// TIA Portal project "Инвинтариаз_V1" (V16)

(* hardware
DEVICE "S7-1200 station_1"  S7-1200 Station
   slot 0: "Rack_0"  S7-1200 Rack  Rack  V1.0
   slot 1: "PLC_1"  CPU 1214C DC/DC/Rly  6ES7 214-1HG40-0XB0  V4.4
   slot 2: "AI 4xRTD_1"  SM 1231 AI4 x RTD  6ES7 231-5PD32-0XB0  V2.0
   slot 3: "AQ 4x14BIT_1"  6ES7 232-4HD32-0XB0  V2.1
*)

// ===== PLC "PLC_1"  CPU 1214C DC/DC/Rly =====

VAR_GLOBAL   // PLC tag table "Default tag table"
   "System_Byte" AT %MB1110 : Byte;
   "FirstScan" AT %M1110.0 : Bool;
   "DiagStatusUpdate" AT %M1110.1 : Bool;
   "AlwaysTRUE" AT %M1110.2 : Bool;
   "AlwaysFALSE" AT %M1110.3 : Bool;
   "Clock_Byte" AT %MB1000 : Byte;
   "Clock_10Hz" AT %M1000.0 : Bool;
   "Clock_5Hz" AT %M1000.1 : Bool;
   "Clock_2.5Hz" AT %M1000.2 : Bool;
   "Clock_2Hz" AT %M1000.3 : Bool;
   "Clock_1.25Hz" AT %M1000.4 : Bool;
   "Clock_1Hz" AT %M1000.5 : Bool;
   "Clock_0.625Hz" AT %M1000.6 : Bool;
   "Clock_0.5Hz" AT %M1000.7 : Bool;
END_VAR

VAR_GLOBAL   // PLC tag table "_Test"
   "Test_En" AT %M0.0 : Bool;
   "t_Lavel_1" AT %M0.1 : Bool;
   "t_Lavel_2" AT %M0.2 : Bool;
   "t_Wardrob1" AT %M0.3 : Bool;
   "t_Wardrob2" AT %M0.4 : Bool;
   "t_time" AT %MD2 : DInt;
   "t_Intemp1" AT %MD6 : Real;
   "t_Intemp_2" AT %MD10 : Real;
   "t_SetTemp" AT %MD14 : Real;
   "t_Set_Delta" AT %MD18 : Real;
   "t_startTime" AT %M0.5 : Bool;
   "t_SetTimer" AT %MD22 : DInt;
   "t_Point_Cold" AT %M0.6 : Bool;
   "t_Finish_Paster" AT %M0.7 : Bool;
   "t_Set_Temp_Cold" AT %MD26 : Real;
   "t_Speed_1" AT %MW30 : Int;
   "t_Speed_2" AT %MW32 : Int;
   "tPaster_St" AT %M1.0 : Bool;
   "tColder_Sr" AT %M1.1 : Bool;
   "t_start" AT %M1.2 : Bool;
   "t_Stop" AT %M1.3 : Bool;
   "t_Alarm" AT %M1.4 : Bool;
END_VAR

TYPE "Tipe_DI"
   STRUCT
      f_DI_out : Bool;
      "bFiltr_on/off" : Bool := true;   // Вкл/выкл фильтрацию входа
      diTime_filtr : Time := T#100ms;   // Уставка времени фильтрации
      bSimulation : Bool;   // Включение режима симуляции
      "bSim_On/Off" : Bool;   // Управление симуляцией
   END_STRUCT;
END_TYPE

DATA_BLOCK "FV_1"   // DB8
{ S7_Optimized_Access := 'FALSE' }
VERSION : 0.1
// stored: InstanceOfName Valve(c/o)
"Valve(c/o)"
BEGIN
END_DATA_BLOCK

DATA_BLOCK "fb_DI_St_DB_1"   // DB9
{ S7_Optimized_Access := 'TRUE' }
VERSION : 0.1
// stored: InstanceOfName fb_DI_St
"fb_DI_St"
BEGIN
END_DATA_BLOCK

DATA_BLOCK "fb_DI_St_DB"   // DB10
{ S7_Optimized_Access := 'TRUE' }
VERSION : 0.1
// stored: InstanceOfName fb_DI_St
"fb_DI_St"
BEGIN
END_DATA_BLOCK

DATA_BLOCK "fb_DI_St_DB_2"   // DB12
{ S7_Optimized_Access := 'TRUE' }
VERSION : 0.1
// stored: InstanceOfName fb_DI_St
"fb_DI_St"
BEGIN
END_DATA_BLOCK

// folder: DB_FB

DATA_BLOCK "Набор Воды_DB"   // DB1
{ S7_Optimized_Access := 'TRUE' }
VERSION : 0.1
// stored: InstanceOfName Набор Воды
"Набор Воды"
BEGIN
END_DATA_BLOCK

DATA_BLOCK "Гл_Блок_Шкафа_DB"   // DB2
{ S7_Optimized_Access := 'TRUE' }
VERSION : 0.1
// stored: InstanceOfName Гл_Блок_Шкафа
"Гл_Блок_Шкафа"
BEGIN
END_DATA_BLOCK

DATA_BLOCK "Контроль темп_DB"   // DB3
{ S7_Optimized_Access := 'TRUE' }
VERSION : 0.1
// stored: InstanceOfName Контроль темп
"Контроль темп"
BEGIN
END_DATA_BLOCK

DATA_BLOCK "Отсчет времени пастеризации_DB"   // DB4
{ S7_Optimized_Access := 'TRUE' }
VERSION : 0.1
// stored: InstanceOfName Отсчет времени пастеризации
"Отсчет времени пастеризации"
BEGIN
END_DATA_BLOCK

DATA_BLOCK "Охлаждение_DB"   // DB6
{ S7_Optimized_Access := 'TRUE' }
VERSION : 0.1
// stored: InstanceOfName Охлаждение
"Охлаждение"
BEGIN
END_DATA_BLOCK

DATA_BLOCK "Старт_DB"   // DB7
{ S7_Optimized_Access := 'TRUE' }
VERSION : 0.1
// stored: InstanceOfName Старт
"Старт"
BEGIN
END_DATA_BLOCK

// folder: HMI

DATA_BLOCK "DI_For_HMI"   // DB11
{ S7_Optimized_Access := 'FALSE' }
VERSION : 0.1
   VAR
      DI_0 : "Tipe_DI";
      DI_1 : "Tipe_DI";
      DI_2 : "Tipe_DI";
      DI_3 : "Tipe_DI";
      DI_4 : "Tipe_DI";
      DI_5 : "Tipe_DI";
      DI_6 : "Tipe_DI";
   END_VAR
BEGIN
END_DATA_BLOCK

// folder: R_trig

DATA_BLOCK "R_trig_Time1S"   // DB5
{ S7_Optimized_Access := 'TRUE' }
VERSION : 0.1
// stored: InstanceOfName R_trig
"R_trig"
BEGIN
END_DATA_BLOCK

// folder: (top level)

FUNCTION_BLOCK "Pump"   // FB1, SCL
{ S7_Optimized_Access := 'FALSE' }
VERSION : 0.1
   VAR_INPUT
      bManualMode : Bool;   // Выбор ручного режима
      bManualStart : Bool;   // Ручной режим - старт
      bManualStop : Bool;   // Ручной режим - стоп
      rManualSpeed : Real;   // Ручной режим - скорость
      bDryRunn : Bool;   // Защита от сухого хода
      bAutoSTop : Bool;   // Остановка насоса
      bAutoStartPerm : Bool;   // Команда на работоу в авто режиме
      rAutoSpeed : Real;   // Скорость в авто режиме
      bАвтоматы : Bool;   // Готовность привода (автоматы)
      bПускатели : Bool;   // Готовность Пускателя
      bDriveRunning : Bool;   // Привод в работе
      bDriveFault : Bool;   // Привод в ошибке
      rMinSpeed : Real;   // Минимальная скорость
      rMaxSpeed : Real := 100.0;   // Максимальная скорость
      bResetFault : Bool;   // Сброс аварии
   END_VAR
   VAR_OUTPUT
      bRunCmd : Bool;   // Пуск частотника
      iSpeedOut : Int;   // Скорость насоса для аналогового выхода
      "rSpeedHMI(0-100)" : Real;   // Скорость работы (0-100) для HMI
      bPumpRunning : Bool;   // Работа
      bPumpFault : Bool;   // Авария
      iStatus : Int;   // Статус (0 - стоп 1 - работа 2 - авария)
   END_VAR
   VAR
      bFaultLatch : Bool;
      bRunRequest : Bool;
      rSpeedPump : Real;   // Скорость насоса
      TON_NotStartRun : TON_TIME;   // ТАймер ожидания сигнала о запуске
      TON_NotContactRun : TON_TIME;   // ТАймер ожидания с контактора
      TON_DryRun : TON_TIME;   // Таймер сухого хода
   END_VAR
BEGIN
   (*
   // 1. Обработка аварий
   // Обработка ожидания сигнала о работе после старта
   IF #bAutoStartPerm THEN
       ;

   END_IF;
   *)

   // 1 Ручной режим
   IF #bManualMode THEN
       // Ручной режим
       IF #bManualStart AND NOT #bManualStop THEN
           #bRunRequest := TRUE;
       ELSIF #bManualStop THEN // OR NOT #bАвтоматы THEN
           #bRunRequest := FALSE;
       END_IF;
   ELSE
       // Автоматический режим
       // 
       //Обработка аварий
       //
       //Таймер ожидания останова по сухому ходу
       #TON_DryRun(IN := NOT #bDryRunn,
                   PT := t#1s);    //
       //--------------------------------------------------------------------------------------------------------
       IF #bAutoStartPerm AND NOT #bAutoSTop AND #bDryRunn THEN
           #TON_NotStartRun(IN := NOT #bDriveRunning AND #bDryRunn, PT := t#5s);  //Таймер ожидания сигнала подтверждения пуска от частотника
           #TON_NotContactRun(IN := NOT #bПускатели, PT := t#10s);  //Таймер ожидания сигнала подтверждения пуска от пускателя


       ELSE
           #TON_NotStartRun(IN :=FALSE,PT := t#5s);
           #TON_NotContactRun(IN := FALSE,PT := t#5s);
       END_IF;
       #bFaultLatch := #TON_NotStartRun.Q OR #TON_NotContactRun.Q OR (#bDriveFault OR NOT #bАвтоматы) OR (NOT #bResetFault AND #bFaultLatch); //Разкоментировать если нужна будет фиксация АЛАРМА, сброс только по входу РЕСЕТ
       #bPumpFault := #bFaultLatch;

       //Старт--------------------------------
       #bRunRequest := #bAutoStartPerm AND NOT #bPumpFault AND NOT #TON_DryRun.Q;
   END_IF;

   // 3. Задание скорости
   IF #bManualMode THEN
       #"rSpeedHMI(0-100)" := LIMIT(MN := #rMinSpeed, IN := #rManualSpeed, MX := #rMaxSpeed);
   ELSE
       #"rSpeedHMI(0-100)" := LIMIT(MN := #rMinSpeed, IN := #rAutoSpeed, MX := #rMaxSpeed);
   END_IF;

   // Преобразование значения от 0-100 до 0-27648 для аналогового выхода
   #iSpeedOut := REAL_TO_INT((#"rSpeedHMI(0-100)"/ 100.0) * 27648.0);

   // 4. Выходные команды и статусы
   // Команды старт
   #bRunCmd := #bRunRequest;

   //Выход статуса для HMI
   #bPumpRunning := #bDriveRunning AND #bRunCmd AND NOT #bAutoSTop OR (#bManualStart AND #bManualMode);



   // 5. Числовой статус (для HMI/SCADA)
   IF #bFaultLatch THEN
       #iStatus := 2; // Авария
   ELSIF #bPumpRunning THEN
       #iStatus := 1; // Работа
   ELSE
       #iStatus := 0; // Стоп
   END_IF;

   IF #bAutoSTop AND NOT #bManualMode THEN
       #bRunCmd := FALSE;
   END_IF;
END_FUNCTION_BLOCK

FUNCTION_BLOCK "Гл_Блок_Шкафа"   // FB2, SCL
{ S7_Optimized_Access := 'TRUE' }
VERSION : 0.1
   VAR_INPUT
      bEn_1 : Bool;   // Разрешение на работу
      bWork_Wardrobe_1 : Bool;   // Выбрана работа шкаф - 1
      bWork_Wardrobe_2 : Bool;   // Выбрана работа шкаф - 2
      iSpeedPump_1 : Int;   // Скорость насоса -1 шкаф
      iSpeedPump_2 : Int;   // Скорость насоса -2 шкаф
      rSetTempPaster : Real;   // Уставка для клапана режим Пастер
      rSetTempColder : Real;   // Уставка для клапана режим Охлаждение
      bPaster : Bool;   // Работа пастеризации
      bColder : Bool;   // Работа охлаждения
   END_VAR
   VAR_OUTPUT
      bValue_2 : Bool;
      bValue_3 : Bool;
      bValue_4 : Bool;
      bValue_5 : Bool;
      bValue_6 : Bool;
      bValue_7 : Bool;
      bPump : Bool;
      iSpeedPump : Int;   // Скорость насоса
      rSetTempPID : Real;   // Уставка для ПИД клапана
   END_VAR
BEGIN

   IF NOT #bEn_1 THEN
       #iSpeedPump := 0;
       #rSetTempPID := 0;

       #bPump := FALSE;
       #bValue_2 := FALSE;
       #bValue_3 := FALSE;
       #bValue_4 := FALSE;
       #bValue_5 := FALSE;
       #bValue_6 := FALSE;
       #bValue_7 := FALSE;

       RETURN;
   END_IF;


   REGION Насос
       //==============Скорость для насоса//==============
       //
       IF #bWork_Wardrobe_2 AND #bWork_Wardrobe_1 THEN
           #iSpeedPump := #iSpeedPump_2;
       ELSIF #bWork_Wardrobe_1 OR #bWork_Wardrobe_2 THEN
           #iSpeedPump := #iSpeedPump_1;
       END_IF;
       //===================================================
       // 
       //==============Старт насоса//==============
       //
       #bPump := TRUE;
       //===================================================
       // 

   END_REGION


   REGION FV-2/3/4/5 - PID


      //////==============Клапана подачи пара ////==============
       #bValue_4 := #bPaster AND NOT #bColder;
       #bValue_5 := #bPaster AND NOT #bColder;
       //======================================================================

       //////==============Клапана подачи холодной воды ////==============
       #bValue_2 := #bColder AND NOT #bPaster;
       #bValue_3 := #bColder AND NOT #bPaster;
       //======================================================================

           ////==============Температура для ПИД регулятора//==============
       IF #bPaster THEN
           #rSetTempPID := #rSetTempPaster;
       ELSIF #bColder THEN
           #rSetTempPID := #rSetTempColder;
       END_IF;
       //======================================================================

   END_REGION


   REGION FV-6/7

       ////==============Управление клапанами подачи в шкафы//==============
       //

       #bValue_6 := #bWork_Wardrobe_1;

       #bValue_7 := #bWork_Wardrobe_2;

       //===================================================
   END_REGION
END_FUNCTION_BLOCK

FUNCTION_BLOCK "Valve(c/o)"   // FB3, SCL
{ S7_Optimized_Access := 'FALSE' }
VERSION : 0.1
   VAR_INPUT
      bAuto_OpenCmd : Bool;   // Команда открыть (автомат)
      bManualMode : Bool;   // Ручной режим (TRUE)
      bManualOpen : Bool;   // Команда открыть в ручном режиме
      bFeedbackOpen : Bool;   // Обратная связь "Открыт"
      tMaxTime : Time;   // Время на открытие
      bResetAlarm : Bool;   // Сброс аварии
      bHaveFeedback : Bool;   // Есть ли обратная связь (0 - нет, 1 есть)
   END_VAR
   VAR_OUTPUT
      bValveOpen : Bool;   // Управляющий выход
      iValveState : Int;   // 0 = Закрыт, 1 = Открыт, 2 = Авария
      bValveFault : Bool;   // Авария
   END_VAR
   VAR
      tiOpenTimer : TON_TIME;   // Таймер на открытие
      bWaitingOpen : Bool;   // Флаг ожидания открытия
      bEnableTimer : Bool;   // Флаг активации таймера
   END_VAR
BEGIN

   // Обновление таймера — всегда в одном месте, вне условий
   #tiOpenTimer(
                IN := #bEnableTimer,
                PT := #tMaxTime
   );

   // Сброс
   IF #bResetAlarm THEN
       #bValveFault := FALSE;
       #bWaitingOpen := FALSE;
       #bEnableTimer := FALSE;
   END_IF;

   // === Режим: РУЧНОЙ ===
   IF #bManualMode THEN
       #bValveOpen := #bManualOpen;
       #bValveFault := FALSE;          // Аварии в ручном режиме не учитываются
       #bEnableTimer := FALSE;
       #bWaitingOpen := FALSE;

       // === Режим: АВТО ===
   ELSE

           // Управление выходом с учетом аварии, с контролем обратной связи
        IF #bAuto_OpenCmd AND NOT #bValveFault THEN
                   #bValveOpen := TRUE;
        ELSE
                   #bValveOpen := FALSE;
               END_IF;

               //  Проверяем, есть ли контроль обратной связи
        IF #bHaveFeedback THEN
            // Контроль открытия
            IF #bAuto_OpenCmd AND NOT #bFeedbackOpen AND NOT #bValveFault THEN
                #bEnableTimer := TRUE;
                #bWaitingOpen := TRUE;
            ELSE
                #bEnableTimer := FALSE;
                ;
                IF #bFeedbackOpen THEN
                    #bWaitingOpen := FALSE;
                END_IF;
            END_IF;
        END_IF;


           // Авария
           IF #tiOpenTimer.Q AND #bWaitingOpen THEN
               #bValveFault := TRUE;
               #bWaitingOpen := FALSE;
           END_IF;

   END_IF;


   // Состояние клапана
   IF #bValveFault THEN
       #iValveState := 2;       // Авария
   ELSIF #bHaveFeedback AND #bFeedbackOpen  THEN
       #iValveState := 1;       // Открыт
   ELSIF NOT #bHaveFeedback AND (NOT #bManualMode AND #bAuto_OpenCmd) OR (#bManualOpen AND #bManualMode) THEN
       #iValveState := 1;       // Открыт 
   ELSE
       #iValveState := 0;       // Закрыт
   END_IF;
END_FUNCTION_BLOCK

FUNCTION_BLOCK "Valve(regul)"   // FB4, SCL
{ S7_Optimized_Access := 'FALSE' }
VERSION : 0.1
   VAR_INPUT
      bManualMode : Bool;   // TRUE = ручной режим, FALSE = автоматический режим
      rAutoSetpoint : Real;   // Уставка открытия клапана в % (0.0–100.0) в автомате
      "bAutoOpen/Close" : Bool;   // Выход Do в автоматическом режиме
      rManualSetpoint : Real;   // Уставка открытия клапана в % (0.0–100.0) в ручном режиме
      "bManualOpen/Close" : Bool;   // Управление выходом открыть/закрыть
   END_VAR
   VAR_OUTPUT
      iAnalogOutput : Int;   // Значение для аналогового выхода (0–27648)
      rValvePosPercent : Real;   // Текущее % открытия клапана для HMI
      bStatusValveOpen : Int;   // Статус сигнал "клапан открыт" (TRUE, если >0%)
      "bOut_Open/Close" : Bool;   // выход для открытия клапана
   END_VAR
   VAR
      rSetpointPercent : Real;   // Расчётная уставка % открытия в текущем режиме
   END_VAR
BEGIN
       // Выбор уставки в зависимости от режима
       IF #bManualMode THEN
           #rSetpointPercent := #rManualSetpoint;
           #"bOut_Open/Close" := #"bManualOpen/Close";
       ELSE
           #rSetpointPercent := #rAutoSetpoint;
           #"bOut_Open/Close" := #"bAutoOpen/Close";
       END_IF;

       // Ограничение % от 0.0 до 100.0
       IF #rSetpointPercent < 0.0 THEN
           #rSetpointPercent := 0.0;
       ELSIF #rSetpointPercent > 100.0 THEN
           #rSetpointPercent := 100.0;
       END_IF;

       // Перевод % в значение для аналогового выхода
       #iAnalogOutput := REAL_TO_INT((#rSetpointPercent / 100.0) * 27648.0);

           // Вывод значения для HMI
       #rValvePosPercent := #rSetpointPercent;

       // Статус клапана для Панели HMI
       IF #rSetpointPercent > 0.0 AND #"bOut_Open/Close" THEN
           #bStatusValveOpen := 1;
       ELSE
           #bStatusValveOpen := 0;
       END_IF;
       ;
END_FUNCTION_BLOCK

FUNCTION_BLOCK "Набор Воды"   // FB5, SCL
{ S7_Optimized_Access := 'TRUE' }
VERSION : 0.1
   VAR_INPUT
      En_1 : Bool;   // разрешение на работу
      bLavel1 : Bool;   // Сработал датчик уровня 1
      bLavel2 : Bool;   // Сработал датчик уровня 2
      bWork_Wardrobe_1 : Bool;   // Выбрана работа шкаф - 1
      bWork_Wardrobe_2 : Bool;   // Выбрана работа шкаф - 2
      diTimeWaitingClose : DInt;   // Время задержки закрытия клапана, сек
   END_VAR
   VAR_OUTPUT
      Value : Bool;   // Работа клапана наполнения
   END_VAR
   VAR
      TON_CloseValve : TON_TIME;
      bStatusValue : Bool;
   END_VAR
   VAR_TEMP
      TimeWaiting : DInt;
   END_VAR
BEGIN
   //Рабоатет блок только при En
   //
   IF NOT #En_1 THEN
       RETURN;
   END_IF;


   REGION TimeWaiting
       // //Время задержки в секундыS
       #TimeWaiting := #diTimeWaitingClose * 1000;

   END_REGION

           //Работа блока обработки наполнения емкости
   //Закрываем клапан по умолчанию
   //
   #TON_CloseValve(IN:=TRUE,
                   PT:=#TimeWaiting);

   IF #TON_CloseValve.Q THEN
       #bStatusValue := FALSE;
   END_IF;

       IF #bWork_Wardrobe_1 AND NOT #bLavel1 THEN
           #bStatusValue := TRUE;
           #TON_CloseValve(IN:=FALSE,
                           PT:=#TimeWaiting);

       ELSIF #bWork_Wardrobe_2 AND NOT #bLavel2 THEN
           #bStatusValue := TRUE;
           #TON_CloseValve(IN := FALSE,
                           PT := #TimeWaiting);
       END_IF;

       #Value := #bStatusValue;
END_FUNCTION_BLOCK

FUNCTION_BLOCK "Контроль темп"   // FB6, SCL
{ S7_Optimized_Access := 'TRUE' }
VERSION : 0.1
   VAR_INPUT
      bEn_1 : Bool;
      bWork_Wardrobe_1 : Bool;   // Выбрана работа шкаф - 1
      bWork_Wardrobe_2 : Bool;   // Выбрана работа шкаф - 2
      rInTemp_1 : Real;   // Входная температура продукта 1
      rInTemp_2 : Real;   // Входная температура продукта 2
      rSetTempProduct : Real;   // Уставка температуры продукта
      rSetDeltaTemp : Real;   // Уставка дельты отклонения температуры
   END_VAR
   VAR_OUTPUT
      bReadyTemps : Bool;   // ВЫход маркер готовности температур
   END_VAR
   VAR_TEMP
      bReadyTemp : Bool;   // Перем для готовности темп
   END_VAR
BEGIN
   //Проверка разраешения выполнения блока
   IF NOT #bEn_1 THEN

       #bReadyTemps := FALSE;
       RETURN;

   END_IF;

   //Сравниваем температуры

   IF #bWork_Wardrobe_1 AND #bWork_Wardrobe_2 THEN
       #bReadyTemp := (#rInTemp_1 >= #rSetTempProduct - #rSetDeltaTemp) AND (#rInTemp_2 >= #rSetTempProduct - #rSetDeltaTemp);
   ELSIF #bWork_Wardrobe_1 THEN
       #bReadyTemp := (#rInTemp_1 >= #rSetTempProduct - #rSetDeltaTemp);
   ELSIF #bWork_Wardrobe_2 THEN
       #bReadyTemp := (#rInTemp_2 >= #rSetTempProduct - #rSetDeltaTemp);
   END_IF;

   // Записываем результат в выход
   // 
   #bReadyTemps := #bReadyTemp;
END_FUNCTION_BLOCK

FUNCTION_BLOCK "Отсчет времени пастеризации"   // FB7, SCL
{ S7_Optimized_Access := 'TRUE' }
VERSION : 0.1
   VAR_INPUT
      bEn_1 : Bool;   // Работа блока
      bStartTaimer : Bool;   // Разрешение на отсчет
      tInSetTime : DInt;   // Заданное время в мин
   END_VAR
   VAR_OUTPUT
      bPasterWorking : Bool;   // Флаг работы пастера
      bFinishTime : Bool;   // Флан финиш таймер
      uiMin : UInt;   // Осталось минут
      uiSec : UInt;   // Осталось сек
   END_VAR
   VAR
      tInToMin : UInt;   // мин, Входное значе
      tInToSec : UInt;   // сек, Входное знач
      tLeftTime : UInt;   // сек, Оставшееся время
      sec : UInt;
   END_VAR
BEGIN
   IF NOT #bEn_1 THEN
       #bPasterWorking := FALSE;
       #bFinishTime := FALSE;
       #uiMin := 0;
       #uiSec := 0;
       #sec := 0;
       #tLeftTime := 0;
       RETURN;
   END_IF;


   REGION Time TO MIN/Sec
       //Переводим введеное значение таймера

       #tInToSec := #tInSetTime * 60; //заданное время в сек
   END_REGION


   //Флаг работы пастера в режиме нагрев и выдержка
   //
   #bPasterWorking := NOT #bFinishTime;

   "R_trig_Time1S"(In:="Clock_5Hz");


   IF #bStartTaimer THEN
       IF "R_trig_Time1S".Q AND NOT (#tLeftTime = 0)  THEN
           #sec := #sec + 1;
       END_IF;
       #tLeftTime := #tInToSec - #sec;
   END_IF;

   IF #bStartTaimer AND (#tLeftTime = 0) THEN
       #bFinishTime := TRUE;
   END_IF;

   #uiMin := #tLeftTime / 60;
   #uiSec := #tLeftTime MOD 60;
END_FUNCTION_BLOCK

FUNCTION_BLOCK "Охлаждение"   // FB8, SCL
{ S7_Optimized_Access := 'TRUE' }
VERSION : 0.1
   VAR_INPUT
      bEn_1 : Bool;
      bWork_Wardrobe_1 : Bool;   // Выбрана работа шкаф - 1
      bWork_Wardrobe_2 : Bool;   // Выбрана работа шкаф - 2
      bPoint_Colder : Bool;   // Выбран режим охлаждения
      bStartColder : Bool;   // Сигнал разрешения на охлаждение
      rSetTempColder : Real;   // Уставка охлаждения
      rInTemp_1 : Real;   // Входная температура Шкаф_1
      rInTemp_2 : Real;   // Входная температура Шкаф_2
   END_VAR
   VAR_OUTPUT
      bCold_Working : Bool;   // Работа режима охлаждения
      bCold_Finish : Bool;   // Финиш охлаждения
   END_VAR
BEGIN
   IF NOT #bEn_1 THEN
       #bCold_Working := FALSE;
       #bCold_Finish := FALSE;
       RETURN;

   END_IF;

   //Проверяем выбор шкафа и разрешение на охлаждение, так же смотрим разрешение на старт работы охлаждения
   //
   IF #bPoint_Colder AND #bStartColder THEN

       #bCold_Working := NOT #bCold_Finish;

       IF #bWork_Wardrobe_1 AND #bWork_Wardrobe_2 THEN

           #bCold_Finish := (#rInTemp_1 <= #rSetTempColder) AND (#rInTemp_2 <= #rSetTempColder);

       ELSIF #bWork_Wardrobe_1 THEN

           #bCold_Finish := (#rInTemp_1 <= #rSetTempColder);

       ELSIF #bWork_Wardrobe_2 THEN

           #bCold_Finish := (#rInTemp_2 <= #rSetTempColder);

       END_IF;
   END_IF;
END_FUNCTION_BLOCK

FUNCTION_BLOCK "Старт"   // FB9, SCL
{ S7_Optimized_Access := 'TRUE' }
VERSION : 0.1
   VAR_INPUT
      bStart : Bool;
      bStop : Bool;
      bAlarm : Bool;
   END_VAR
   VAR_OUTPUT
      bWorkingMode : Bool;
   END_VAR
   VAR
      fb_Start : "R_trig";
      fb_Stop : "R_trig";
   END_VAR
BEGIN

   REGION r_trigers
       // обработка сигналов
       #fb_Start(In:=#bStart);
       #fb_Stop(In:=#bStop);
   END_REGION



   IF #fb_Start.Q AND NOT #bAlarm THEN
       #bWorkingMode := true;
   END_IF;

   IF #bAlarm THEN
       #bWorkingMode := FALSE;
   END_IF;

   IF #fb_Stop.Q THEN
       #bWorkingMode := FALSE;
   END_IF;
END_FUNCTION_BLOCK

FUNCTION_BLOCK "FB_Аварии"   // FB10, SCL
{ S7_Optimized_Access := 'FALSE' }
VERSION : 0.1
   VAR_INPUT
      Rtrig_Reset : Bool;
   END_VAR
   VAR_OUTPUT
      ALARM_Active : Bool;   // Флаг активной аварии
   END_VAR
   VAR
      LatchedEmergency : Bool;   // Зафиксированная аварийная ситуация
      bAlarmAvtomats : Bool;   // Авария автоматов
      bAlarmAI : Bool;   // Авария аналоговых датчиков
      bAlarmPumps : Bool;   // Авария насосов
      bAlarmConveyors : Bool;   // Авария Конвейеров
      bAlarmFVs : Bool;   // Авария клапанов
      bAlarmDI_all : Bool;   // Авария по дискретным входам "общая"
      bAlarmLowLevel : Bool;   // Авария по низкому уровню емкостей
      bAlarmProcess : Bool;   // Аварии которые возникают в результате работы
      mReset : Bool;
      TON_LowLevel : TON_TIME;   // Таймер для аварийного уровня емкостей
      bResetaALARM : Bool;   // Сброс аварии (кнопка на панели/системе)
   END_VAR
   VAR_TEMP
      nAi : Int;
      nPump : Int;
      nConv : Int;
      nFV : Int;
      nAvtomat : Int;
      numPump : Int;
   END_VAR
BEGIN
   REGION Предварительное отрицание
       // Сброс в 0 при отсутсвии аварий для цикла и массивов
       #bAlarmAvtomats := FALSE;
       #bAlarmAI := FALSE;
       #bAlarmPumps := FALSE;
       #bAlarmConveyors := FALSE;
       #bAlarmFVs := FALSE;


   END_REGION



   //Авария аналоговых входов
   //--------------------------


   //Авария НАСОСОВ
   //--------------------------



   //Авария Клапанов
   //--------------------------


   //Авария по входам DI
   //---------------------------



   //Обработка всех аварий с выводом сигнала наличия АВАРИЯ
   //----------------------------------------------------------------
                       IF #bAlarmAI OR #bAlarmPumps OR #bAlarmFVs OR #bAlarmDI_all OR #bAlarmProcess THEN

                           #ALARM_Active := TRUE;

                       END_IF;



   //Отлавливаем фронт Ресета....................................
   (*
   #bResetaALARM := #Rtrig_Reset AND NOT #mReset;
   #mReset := #Rtrig_Reset;
   *)

    //Если нужен жесткий сбро, игнорирует все аварии                      
   #bResetaALARM := #Rtrig_Reset;

   //-------------------------------------------------------------                       
                          // Сброс аварии
   IF #bResetaALARM THEN
       #ALARM_Active := FALSE;
   END_IF;
END_FUNCTION_BLOCK

FUNCTION_BLOCK "fb_DI_St"   // FB11, SCL
{ S7_Optimized_Access := 'TRUE' }
VERSION : 0.1
   VAR_INPUT
      In : Bool;
   END_VAR
   VAR_OUTPUT
      f_Di_Out : Bool;
   END_VAR
   VAR_IN_OUT
      Type_DI : "Tipe_DI";
   END_VAR
   VAR
      aTON_Filtr : TON_TIME;   // Следить за кол-вом DI
      bTonIn : Bool;
      Volue : Bool;
   END_VAR
   VAR_TEMP
      i : Int;
      SizeArreyUp : Int;   // Размер массива
      SizeArreyDown : Int;
   END_VAR
   VAR CONSTANT
      n : Int := 10;
   END_VAR
BEGIN

       REGION Таймер фильтрации входа
           // управление таймером 
           #bTonIn := NOT #Type_DI.bSimulation AND #Type_DI."bFiltr_on/off" AND #In;
           // вызов таймера фильтрации
           #aTON_Filtr(IN := #bTonIn,
                       PT := #Type_DI.diTime_filtr);
       END_REGION



       //-------------Условие симуляции, если да работает только по сигналам симулирования 
       IF (#Type_DI.bSimulation = TRUE) THEN
           #Volue := #Type_DI."bSim_On/Off";

       //------------Условие если фильтрация включена--------------------
       ELSIF #Type_DI."bFiltr_on/off" = TRUE THEN

           #Volue := #aTON_Filtr.Q;    //Выход по таймеру значения таймера

       ELSE
           #Volue := #In;

       END_IF;

       //Присвоение выходу значения
       #Type_DI.f_DI_out :=  #Volue;
       #f_Di_Out := #Volue;
END_FUNCTION_BLOCK

FUNCTION "Клапан О/З" : Void   // FC1, LAD
{ S7_Optimized_Access := 'TRUE' }
VERSION : 0.1
BEGIN

REGION Network 1
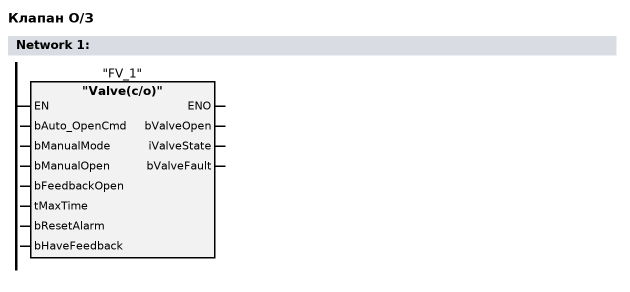
   RUNG wire#powerrail
      "FV_1"(bAuto_OpenCmd :=, bManualMode :=, bManualOpen :=, bFeedbackOpen :=, tMaxTime :=, bResetAlarm :=, bHaveFeedback :=, bValveOpen =>, iValveState =>, bValveFault =>)
   END_RUNG
   // the same network as SCL:
   "FV_1"();   // "Valve(c/o)"
END_REGION
END_FUNCTION

FUNCTION "DI" : Void   // FC2, LAD
{ S7_Optimized_Access := 'TRUE' }
VERSION : 0.1
BEGIN

REGION Network 1
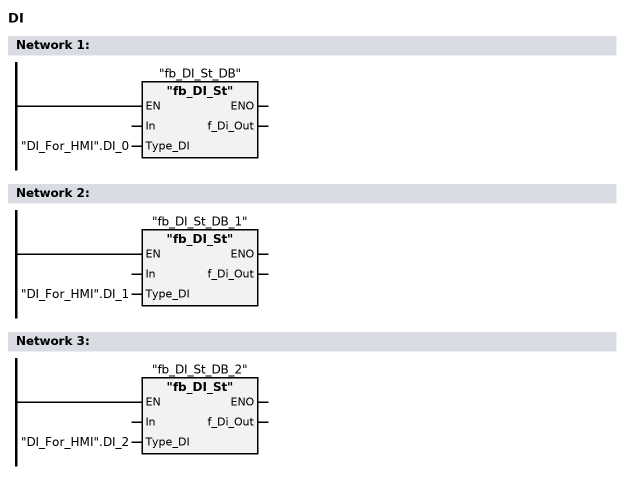
   RUNG wire#powerrail
      "fb_DI_St_DB"(In :=, Type_DI := "DI_For_HMI".DI_0, f_Di_Out =>)
   END_RUNG
   // the same network as SCL:
   "fb_DI_St_DB"(Type_DI := "DI_For_HMI".DI_0);   // "fb_DI_St"
END_REGION

REGION Network 2
   RUNG wire#powerrail
      "fb_DI_St_DB_1"(In :=, Type_DI := "DI_For_HMI".DI_1, f_Di_Out =>)
   END_RUNG
   // the same network as SCL:
   "fb_DI_St_DB_1"(Type_DI := "DI_For_HMI".DI_1);   // "fb_DI_St"
END_REGION

REGION Network 3
   RUNG wire#powerrail
      "fb_DI_St_DB_2"(In :=, Type_DI := "DI_For_HMI".DI_2, f_Di_Out =>)
   END_RUNG
   // the same network as SCL:
   "fb_DI_St_DB_2"(Type_DI := "DI_For_HMI".DI_2);   // "fb_DI_St"
END_REGION
END_FUNCTION

FUNCTION "Все в Авто" : Void   // FC12, SCL
{ S7_Optimized_Access := 'TRUE' }
VERSION : 0.1
BEGIN
END_FUNCTION

FUNCTION "RestetAlarms" : Void   // FC13, SCL
{ S7_Optimized_Access := 'TRUE' }
VERSION : 0.1
BEGIN
END_FUNCTION

ORGANIZATION_BLOCK "Main"   // OB1, LAD, ProgramCycle
TITLE = "Main Program Sweep (Cycle)"
{ S7_Optimized_Access := 'TRUE' }
VERSION : 0.1
BEGIN

REGION Network 2: Старт работы
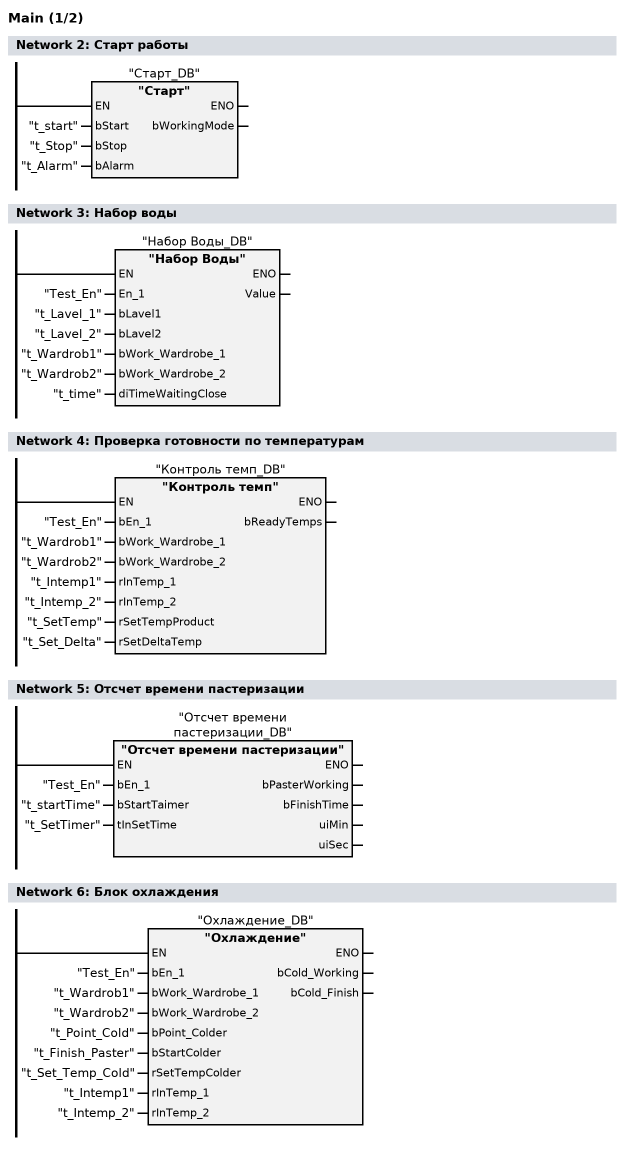
   RUNG wire#powerrail
      "Старт_DB"(bStart := "t_start", bStop := "t_Stop", bAlarm := "t_Alarm", bWorkingMode =>)
   END_RUNG
   // the same network as SCL:
   "Старт_DB"(bStart := "t_start", bStop := "t_Stop", bAlarm := "t_Alarm");   // "Старт"
END_REGION

REGION Network 3: Набор воды
   RUNG wire#powerrail
      "Набор Воды_DB"(En_1 := "Test_En", bLavel1 := "t_Lavel_1", bLavel2 := "t_Lavel_2", bWork_Wardrobe_1 := "t_Wardrob1", bWork_Wardrobe_2 := "t_Wardrob2", diTimeWaitingClose := "t_time", Value =>)
   END_RUNG
   // the same network as SCL:
   "Набор Воды_DB"(En_1 := "Test_En",   // "Набор Воды"
                   bLavel1 := "t_Lavel_1",
                   bLavel2 := "t_Lavel_2",
                   bWork_Wardrobe_1 := "t_Wardrob1",
                   bWork_Wardrobe_2 := "t_Wardrob2",
                   diTimeWaitingClose := "t_time");
END_REGION

REGION Network 4: Проверка готовности по температурам
   RUNG wire#powerrail
      "Контроль темп_DB"(bEn_1 := "Test_En", bWork_Wardrobe_1 := "t_Wardrob1", bWork_Wardrobe_2 := "t_Wardrob2", rInTemp_1 := "t_Intemp1", rInTemp_2 := "t_Intemp_2", rSetTempProduct := "t_SetTemp", rSetDeltaTemp := "t_Set_Delta", bReadyTemps =>)
   END_RUNG
   // the same network as SCL:
   "Контроль темп_DB"(bEn_1 := "Test_En",   // "Контроль темп"
                      bWork_Wardrobe_1 := "t_Wardrob1",
                      bWork_Wardrobe_2 := "t_Wardrob2",
                      rInTemp_1 := "t_Intemp1",
                      rInTemp_2 := "t_Intemp_2",
                      rSetTempProduct := "t_SetTemp",
                      rSetDeltaTemp := "t_Set_Delta");
END_REGION

REGION Network 5: Отсчет времени пастеризации
   RUNG wire#powerrail
      "Отсчет времени пастеризации_DB"(bEn_1 := "Test_En", bStartTaimer := "t_startTime", tInSetTime := "t_SetTimer", bFinishTime =>, uiMin =>, uiSec =>, bPasterWorking =>)
   END_RUNG
   // the same network as SCL:
   "Отсчет времени пастеризации_DB"(bEn_1 := "Test_En",   // "Отсчет времени пастеризации"
                           bStartTaimer := "t_startTime",
                           tInSetTime := "t_SetTimer");
END_REGION

REGION Network 6: Блок охлаждения
   RUNG wire#powerrail
      "Охлаждение_DB"(bEn_1 := "Test_En", bWork_Wardrobe_1 := "t_Wardrob1", bWork_Wardrobe_2 := "t_Wardrob2", bPoint_Colder := "t_Point_Cold", bStartColder := "t_Finish_Paster", rSetTempColder := "t_Set_Temp_Cold", rInTemp_1 := "t_Intemp1", rInTemp_2 := "t_Intemp_2", bCold_Working =>, bCold_Finish =>)
   END_RUNG
   // the same network as SCL:
   "Охлаждение_DB"(bEn_1 := "Test_En",   // "Охлаждение"
                   bWork_Wardrobe_1 := "t_Wardrob1",
                   bWork_Wardrobe_2 := "t_Wardrob2",
                   bPoint_Colder := "t_Point_Cold",
                   bStartColder := "t_Finish_Paster",
                   rSetTempColder := "t_Set_Temp_Cold",
                   rInTemp_1 := "t_Intemp1",
                   rInTemp_2 := "t_Intemp_2");
END_REGION

REGION Network 7: Блок работы в авто
   // управление клапанами и уставками
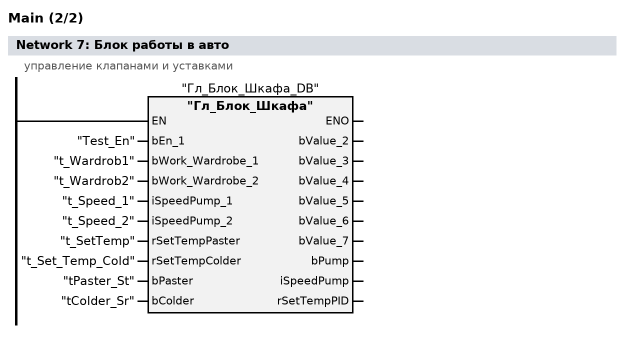
   RUNG wire#powerrail
      "Гл_Блок_Шкафа_DB"(bEn_1 := "Test_En", bWork_Wardrobe_1 := "t_Wardrob1", bWork_Wardrobe_2 := "t_Wardrob2", iSpeedPump_1 := "t_Speed_1", iSpeedPump_2 := "t_Speed_2", rSetTempPaster := "t_SetTemp", rSetTempColder := "t_Set_Temp_Cold", bPaster := "tPaster_St", bColder := "tColder_Sr", bValue_2 =>, bValue_3 =>, bValue_4 =>, bValue_5 =>, bValue_6 =>, bValue_7 =>, bPump =>, iSpeedPump =>, rSetTempPID =>)
   END_RUNG
   // the same network as SCL:
   "Гл_Блок_Шкафа_DB"(bEn_1 := "Test_En",   // "Гл_Блок_Шкафа"
                      bWork_Wardrobe_1 := "t_Wardrob1",
                      bWork_Wardrobe_2 := "t_Wardrob2",
                      iSpeedPump_1 := "t_Speed_1",
                      iSpeedPump_2 := "t_Speed_2",
                      rSetTempPaster := "t_SetTemp",
                      rSetTempColder := "t_Set_Temp_Cold",
                      bPaster := "tPaster_St",
                      bColder := "tColder_Sr");
END_REGION
END_ORGANIZATION_BLOCK

ORGANIZATION_BLOCK "Аварии/Ресет"   // OB123, LAD, ProgramCycle
TITLE = "Main Program Sweep (Cycle)"
{ S7_Optimized_Access := 'TRUE' }
VERSION : 0.1
   VAR_INPUT
      Initial_Call : Bool;   // Initial call of this OB
      Remanence : Bool;   // =True, if remanent data are available
   END_VAR
BEGIN
END_ORGANIZATION_BLOCK

ORGANIZATION_BLOCK "Исполнительные узлы"   // OB124, LAD, ProgramCycle
TITLE = "Main Program Sweep (Cycle)"
{ S7_Optimized_Access := 'TRUE' }
VERSION : 0.1
   VAR_INPUT
      Initial_Call : Bool;   // Initial call of this OB
      Remanence : Bool;   // =True, if remanent data are available
   END_VAR
BEGIN

REGION Network 1: клапана о/з
END_REGION

REGION Network 2: DI
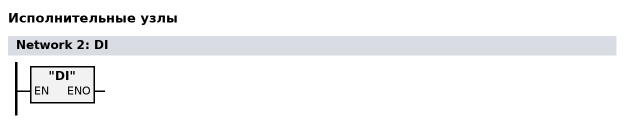
   RUNG wire#powerrail
      "DI"()
   END_RUNG
   // the same network as SCL:
   "DI"();
END_REGION
END_ORGANIZATION_BLOCK

// folder: R_trig

FUNCTION_BLOCK "R_trig"   // FB16, SCL
{ S7_Optimized_Access := 'TRUE' }
VERSION : 0.1
   VAR_INPUT
      In : Bool;
   END_VAR
   VAR_OUTPUT
      Q : Bool;
   END_VAR
   VAR
      Click_M : Bool;
   END_VAR
BEGIN
   #Q := #In AND NOT #Click_M;
   #Click_M := #In;
END_FUNCTION_BLOCK